        // Search power groups from LARGEST to SMALLEST
        FOR g := 1 TO Num_Unique_Powers DO
            Target_Power_Value := Unique_Powers[g];
            
            // Does this power fit?
            IF Target_Power_Value <= Power_Needed THEN
                // Find available step with this power, lowest cycles
                FOR i := 1 TO Number_Of_Steps DO
                    IF Step_Power_Rating[i] = Target_Power_Value THEN
                        Step_Available := NOT Coil_Internal[i] AND NOT Step_Quarantined[i];
                        
                        IF Step_Available AND Step_Cycle_Count[i] < Min_Cycles THEN
                            Best_Step := i;
                            Min_Cycles := Step_Cycle_Count[i];
                        END_IF;
                    END_IF;
                END_FOR;
                
                // Found a step? Use it
                IF Best_Step > 0 THEN
                    EXIT;
                END_IF;
            END_IF;
        END_FOR;
        
        // If no large step fits, find smallest available step
        IF Best_Step = 0 THEN
            FOR g := Num_Unique_Powers TO 1 BY -1 DO
                Target_Power_Value := Unique_Powers[g];
                
                FOR i := 1 TO Number_Of_Steps DO
                    IF Step_Power_Rating[i] = Target_Power_Value THEN
                        Step_Available := NOT Coil_Internal[i] AND NOT Step_Quarantined[i];
                        
                        IF Step_Available THEN
                            IF Best_Step = 0 OR Step_Cycle_Count[i] < Min_Cycles THEN
                                Best_Step := i;
                                Min_Cycles := Step_Cycle_Count[i];
                            END_IF;
                        END_IF;
                    END_IF;
                END_FOR;
                
                IF Best_Step > 0 THEN
                    EXIT;
                END_IF;
            END_FOR;
        END_IF;
        
        // Turn ON selected step
        IF Best_Step > 0 THEN
            Coil_Internal[Best_Step] := TRUE;
            Step_Cycle_Count[Best_Step] := Step_Cycle_Count[Best_Step] + 1;
        END_IF;
        
        Step_Up_Timer(IN := FALSE);
    END_IF;

// ============================================
// NEED TO REMOVE POWER?
// ============================================
ELSIF Power_Needed < -Deadband_kW THEN
    Step_Down_Timer(IN := TRUE, PT := Step_Down_Delay);
    Step_Up_Timer(IN := FALSE);
    
    IF Step_Down_Timer.Q THEN
        Best_Step := 0;
        Max_Cycles := 0;
        
        // Search power groups from SMALLEST to LARGEST
        FOR g := Num_Unique_Powers TO 1 BY -1 DO
            Target_Power_Value := Unique_Powers[g];
            
            // Does this power fit?
            IF Target_Power_Value <= ABS(Power_Needed) THEN
                // Find ON step with this power, highest cycles
                FOR i := 1 TO Number_Of_Steps DO
                    IF Step_Power_Rating[i] = Target_Power_Value AND Coil_Internal[i] THEN
                        IF Step_Cycle_Count[i] >= Max_Cycles THEN
                            Best_Step := i;
                            Max_Cycles := Step_Cycle_Count[i];
                        END_IF;
                    END_IF;
                END_FOR;
                
                IF Best_Step > 0 THEN
                    EXIT;
                END_IF;
            END_IF;
        END_FOR;
        
        // If no step fits, find smallest ON step
        IF Best_Step = 0 THEN
            FOR g := Num_Unique_Powers TO 1 BY -1 DO
                Target_Power_Value := Unique_Powers[g];
                
                FOR i := 1 TO Number_Of_Steps DO
                    IF Step_Power_Rating[i] = Target_Power_Value AND Coil_Internal[i] THEN
                        Best_Step := i;
                        EXIT;
                    END_IF;
                END_FOR;
                
                IF Best_Step > 0 THEN
                    EXIT;
                END_IF;
            END_FOR;
        END_IF;
        
        // Turn OFF selected step
        IF Best_Step > 0 THEN
            Coil_Internal[Best_Step] := FALSE;
        END_IF;
        
        Step_Down_Timer(IN := FALSE);
    END_IF;

ELSE
    // At target - reset timers
    Step_Up_Timer(IN := FALSE);
    Step_Down_Timer(IN := FALSE);
END_IF;

END_IF; // End of non-maintenance mode

// ============================================
// FEEDBACK MONITORING
// ============================================
Any_Feedback_Fault := FALSE;

IF Enable_Feedback_Monitoring THEN
    FOR i := 1 TO Number_Of_Steps DO
        // Reset timer on rising edge (coil just turned ON)
        IF Coil_Internal[i] AND NOT Coil_Prev[i] THEN
            FB_Timer[i](IN := FALSE);
        END_IF;
        
        // Monitor: Coil ON but no feedback
        FB_Timer[i](
            IN := Coil_Internal[i] AND NOT Step_Feedback[i] AND NOT FB_Fault_Latched[i],
            PT := Feedback_Timeout
        );
        
        // Timeout = fault, quarantine step
        IF FB_Timer[i].Q THEN
            FB_Fault_Latched[i] := TRUE;
            Step_Quarantine_Feedback[i] := TRUE;
            Coil_Internal[i] := FALSE;
        END_IF;
        
        IF FB_Fault_Latched[i] THEN
            Any_Feedback_Fault := TRUE;
        END_IF;
        
        Coil_Prev[i] := Coil_Internal[i];
    END_FOR;
END_IF;

// ============================================
// TOTAL POWER MONITORING
// ============================================
IF Enable_Power_Monitoring AND Active_Step_Count > 0 THEN
    // Calculate expected power from ON steps
    Expected_Power := 0.0;
    FOR i := 1 TO Number_Of_Steps DO
        IF Coil_Internal[i] THEN
            Expected_Power := Expected_Power + Step_Power_Rating[i];
        END_IF;
    END_FOR;
    
    // Calculate difference
    Power_Diff := ABS(Measured_Total_Power - Expected_Power);
    
    // Calculate percentage
    IF Expected_Power > 0.0 THEN
        Power_Mismatch_Percent := (Power_Diff / Expected_Power) * 100.0;
    ELSE
        Power_Mismatch_Percent := 0.0;
    END_IF;
    
    // Check if outside tolerance
    Power_Monitor_Timer(
        IN := Power_Mismatch_Percent > Power_Tolerance_Percent,
        PT := Power_Monitor_Delay
    );
    
    IF Power_Monitor_Timer.Q THEN
        Total_Power_Warning := TRUE;
    ELSIF Power_Mismatch_Percent <= Power_Tolerance_Percent THEN
        Total_Power_Warning := FALSE;
        Power_Monitor_Timer(IN := FALSE);
    END_IF;
ELSE
    Power_Monitor_Timer(IN := FALSE);
    Power_Mismatch_Percent := 0.0;
END_IF;

// ============================================
// COPY TO OUTPUT
// ============================================
FOR i := 1 TO LB_NUMBER_OF_STEPS DO
    Step_Coil_Cmd[i] := Coil_Internal[i];
END_FOR;

// ============================================
// CALCULATE RELEASED POWER (final)
// ============================================
Released_Power_kW := 0.0;
Active_Step_Count := 0;
FOR i := 1 TO Number_Of_Steps DO
    IF Coil_Internal[i] THEN
        Released_Power_kW := Released_Power_kW + Step_Power_Rating[i];
        Active_Step_Count := Active_Step_Count + 1;
    END_IF;
END_FOR;

// ============================================
// STATUS MESSAGE
// ============================================
IF Total_Power_Warning THEN
    Status_Text := 'POWER MISMATCH WARNING';
ELSIF Any_Feedback_Fault THEN
    Status_Text := 'FEEDBACK FAULT';
ELSIF Maintenance_Mode THEN
    Status_Text := 'Maintenance mode';
ELSIF At_Target THEN
    Status_Text := 'At target';
ELSIF Power_Needed > 0.0 THEN
    Status_Text := 'Increasing load';
ELSIF Power_Needed < 0.0 THEN
    Status_Text := 'Decreasing load';
ELSE
    Status_Text := 'Ready';
END_IF;

END_FUNCTION_BLOCK

// ---- POUs/FB_Mode_Manager.TcPOU
FUNCTION_BLOCK FB_Mode_Manager
VAR_INPUT
    Mode_Select             : UINT;
    Master_Enable           : BOOL;
    Emergency_Active        : BOOL;
    System_Ready            : BOOL;
END_VAR
VAR_OUTPUT
    Active_Mode             : UINT;
    Mode_Name               : STRING(30);
    Mode_Ready              : BOOL;
    Enable_Output           : BOOL;
END_VAR
VAR
    Mode_Select_Prev        : UINT;
END_VAR

// Emergency forces OFF mode
IF Emergency_Active THEN
    Active_Mode := LB_MODE_OFF;
    Mode_Name := 'EMERGENCY STOP';
    Mode_Ready := FALSE;
    Enable_Output := FALSE;
    RETURN;
END_IF;

// Master enable check
IF NOT Master_Enable THEN
    Active_Mode := LB_MODE_OFF;
    Mode_Name := 'OFF - Enable Required';
    Mode_Ready := FALSE;
    Enable_Output := FALSE;
    RETURN;
END_IF;

// Mode selection
IF Mode_Select <> Mode_Select_Prev THEN
    Active_Mode := Mode_Select;
END_IF;
Mode_Select_Prev := Mode_Select;

// Mode names and enable logic
CASE Active_Mode OF
    LB_MODE_OFF:
        Mode_Name := 'OFF';
        Mode_Ready := TRUE;
        Enable_Output := FALSE;
    
    LB_MODE_AUTO_LEVELING:
        Mode_Name := 'AUTO LOAD LEVELING';
        Mode_Ready := System_Ready;
        Enable_Output := System_Ready;
    
    LB_MODE_NUMERIC:
        Mode_Name := 'NUMERIC LOAD CONTROL';
        Mode_Ready := System_Ready;
        Enable_Output := System_Ready;
    
    LB_MODE_REVERSE_POWER:
        Mode_Name := 'REVERSE POWER';
        Mode_Ready := System_Ready;
        Enable_Output := System_Ready;
    
    LB_MODE_MANUAL:
        Mode_Name := 'MANUAL SWITCH CONTROL';
        Mode_Ready := System_Ready;
        Enable_Output := System_Ready;
    
    LB_MODE_RECIPE:
        Mode_Name := 'RECIPE MODE';
        Mode_Ready := System_Ready;
        Enable_Output := System_Ready;
    
    LB_MODE_MAINTENANCE:
        Mode_Name := 'MAINTENANCE MODE';
        Mode_Ready := TRUE;
        Enable_Output := TRUE;
    
    ELSE
        Mode_Name := 'UNKNOWN MODE';
        Mode_Ready := FALSE;
        Enable_Output := FALSE;
        Active_Mode := LB_MODE_OFF;
END_CASE;

END_FUNCTION_BLOCK

// ---- POUs/FB_DataLogger.TcPOU
FUNCTION_BLOCK FB_DataLogger
(******************************************************************************
 * FB_DataLogger
 * 
 * Purpose: Data logging for Load Bank system
 *   1. Circular buffer for HMI trends (real-time viewing)
 *   2. USB/SD CSV file logging (long-term storage)
 *
 * Features:
 *   - Configurable sample rate (1s to 60s)
 *   - Configurable buffer size (up to 3600 samples)
 *   - Daily CSV files with auto-rotation
 *   - Enable/disable for buffer and USB separately
 *
 * Author: Load Bank Project
 * Date: January 2026
 ******************************************************************************)

VAR_INPUT
    // Enable controls
    Enable                  : BOOL := TRUE;         // Master enable
    USB_Log_Enable          : BOOL := TRUE;         // Enable USB file logging
    
    // Sample rate (from GVL_Persistent)
    Sample_Time             : TIME := T#10s;        // How often to sample
    Buffer_Size             : UINT := 360;          // Active buffer size (max 3600)
    
    // Data inputs - Power
    Power_Released          : REAL;
    Power_Target            : REAL;
    
    // Data inputs - Temperature (up to 4 TCs)
    Temp_TC1                : REAL;
    Temp_TC2                : REAL;
    Temp_TC3                : REAL;
    Temp_TC4                : REAL;
    Number_Of_TCs           : UINT := 2;            // How many TCs configured
    
    // Data inputs - Voltage (3-phase)
    Voltage_L1L2            : REAL;
    Voltage_L2L3            : REAL;
    Voltage_L3L1            : REAL;
    
    // Data inputs - Current (3-phase)
    Current_I1              : REAL;
    Current_I2              : REAL;
    Current_I3              : REAL;
    
    // USB path configuration
    USB_Path                : STRING(100) := 'C:\DataLog\';  // Path for CSV files
    
    // Commands
    Clear_Buffer            : BOOL;                 // Clear all trend buffers
    
END_VAR

VAR_OUTPUT
    // Status
    Buffer_Index            : UINT;                 // Current write position (0 to Buffer_Size-1)
    Buffer_Full             : BOOL;                 // Buffer has wrapped at least once
    Samples_Logged          : UDINT;                // Total samples since enable
    
    // USB status
    USB_Active              : BOOL;                 // USB logging is active
    USB_File_Open           : BOOL;                 // File currently open
    USB_Error               : BOOL;                 // Error writing to USB
    USB_Error_Code          : UDINT;                // Last error code
    Current_File_Name       : STRING(50);           // Current log file name
    
    // Trend buffer outputs (circular buffers)
    // These are written to GVL arrays for HMI access
    Trend_Write_Index       : UINT;                 // Current write index for HMI
    
END_VAR

VAR
    // Timing
    Sample_Timer            : TON;
    Sample_Trigger          : BOOL;
    
    // Buffer management
    Internal_Index          : UINT := 0;
    Buffer_Wrapped          : BOOL := FALSE;
    
    // USB file handling
    FB_FileOpen             : FB_FileOpen;
    FB_FilePuts             : FB_FilePuts;
    FB_FileClose            : FB_FileClose;
    FB_CreateDir            : FB_CreateDir;
    
    File_Handle             : UINT := 0;
    File_State              : UINT := 0;            // State machine for file ops
    Write_Buffer            : STRING(500);          // Line buffer for CSV
    
    // Date tracking for daily files
    Last_Day                : WORD := 0;
    Last_Month              : WORD := 0;
    System_Time             : TIMESTRUCT;
    FB_GetTime              : NT_GetTime;
    
    // Internal flags
    Init_Done               : BOOL := FALSE;
    Dir_Created             : BOOL := FALSE;
    Need_New_File           : BOOL := FALSE;
    Write_Pending           : BOOL := FALSE;
    Close_Pending           : BOOL := FALSE;
    
    // Helpers
    i                       : UINT;
    sTemp                   : STRING(20);
    
END_VAR

VAR CONSTANT
    MAX_BUFFER              : UINT := 3600;         // Maximum array size
END_VAR

// ============================================================================
// INITIALIZATION
// ============================================================================
IF NOT Init_Done THEN
    Internal_Index := 0;
    Buffer_Wrapped := FALSE;
    Samples_Logged := 0;
    File_State := 0;
    Init_Done := TRUE;
END_IF

// ============================================================================
// CLEAR BUFFER COMMAND
// ============================================================================
IF Clear_Buffer THEN
    Internal_Index := 0;
    Buffer_Wrapped := FALSE;
    Samples_Logged := 0;
    
    // Clear all GVL trend arrays
    FOR i := 1 TO MAX_BUFFER DO
        Trend_Power_Released[i] := 0.0;
        Trend_Power_Target[i] := 0.0;
        Trend_Temp_TC1[i] := 0.0;
        Trend_Temp_TC2[i] := 0.0;
        Trend_Temp_TC3[i] := 0.0;
        Trend_Temp_TC4[i] := 0.0;
        Trend_Voltage_L1L2[i] := 0.0;
        Trend_Voltage_L2L3[i] := 0.0;
        Trend_Voltage_L3L1[i] := 0.0;
        Trend_Current_I1[i] := 0.0;
        Trend_Current_I2[i] := 0.0;
        Trend_Current_I3[i] := 0.0;
    END_FOR
END_IF

// ============================================================================
// SAMPLE TIMER
// ============================================================================
Sample_Timer(
    IN := Enable AND NOT Sample_Timer.Q,
    PT := Sample_Time
);

Sample_Trigger := Sample_Timer.Q;

// Reset timer on trigger
IF Sample_Trigger THEN
    Sample_Timer(IN := FALSE);
END_IF

// ============================================================================
// GET CURRENT TIME (for file naming and timestamps)
// ============================================================================
FB_GetTime(
    NETID := '',
    START := TRUE,
    TMOUT := T#1s
);

IF NOT FB_GetTime.BUSY AND NOT FB_GetTime.ERR THEN
    System_Time := FB_GetTime.TIMESTR;
END_IF

// ============================================================================
// DATA SAMPLING - CIRCULAR BUFFER
// ============================================================================
IF Enable AND Sample_Trigger THEN
    
    // Clamp buffer size
    IF Buffer_Size > MAX_BUFFER THEN
        Buffer_Size := MAX_BUFFER;
    END_IF
    IF Buffer_Size < 1 THEN
        Buffer_Size := 1;
    END_IF
    
    // Calculate array index (1-based for TwinCAT arrays)
    i := Internal_Index + 1;
    
    // Write to GVL trend arrays
    Trend_Power_Released[i] := Power_Released;
    Trend_Power_Target[i] := Power_Target;
    Trend_Temp_TC1[i] := Temp_TC1;
    Trend_Temp_TC2[i] := Temp_TC2;
    Trend_Temp_TC3[i] := Temp_TC3;
    Trend_Temp_TC4[i] := Temp_TC4;
    Trend_Voltage_L1L2[i] := Voltage_L1L2;
    Trend_Voltage_L2L3[i] := Voltage_L2L3;
    Trend_Voltage_L3L1[i] := Voltage_L3L1;
    Trend_Current_I1[i] := Current_I1;
    Trend_Current_I2[i] := Current_I2;
    Trend_Current_I3[i] := Current_I3;
    
    // Increment index with wrap-around
    Internal_Index := Internal_Index + 1;
    IF Internal_Index >= Buffer_Size THEN
        Internal_Index := 0;
        Buffer_Wrapped := TRUE;
    END_IF
    
    // Update outputs
    Buffer_Index := Internal_Index;
    Buffer_Full := Buffer_Wrapped;
    Samples_Logged := Samples_Logged + 1;
    Trend_Write_Index := Internal_Index;
    
    // Trigger USB write
    IF USB_Log_Enable THEN
        Write_Pending := TRUE;
    END_IF
    
END_IF

// ============================================================================
// USB FILE LOGGING - STATE MACHINE
// ============================================================================
IF USB_Log_Enable AND Enable THEN
    
    CASE File_State OF
        
        // --------------------------------------------------------------------
        // State 0: Idle / Check if new file needed
        // --------------------------------------------------------------------
        0:
            USB_Active := TRUE;
            
            // Check if date changed (need new daily file)
            IF (System_Time.wDay <> Last_Day) OR (System_Time.wMonth <> Last_Month) OR NOT USB_File_Open THEN
                Need_New_File := TRUE;
                
                // Close existing file first if open
                IF USB_File_Open THEN
                    File_State := 50;  // Go to close state
                ELSE
                    File_State := 10;  // Go to create directory
                END_IF
            ELSIF Write_Pending THEN
                File_State := 30;  // Go to write state
            END_IF
            
        // --------------------------------------------------------------------
        // State 10: Create directory if needed
        // --------------------------------------------------------------------
        10:
            FB_CreateDir(
                sNetId := '',
                sPathName := USB_Path,
                ePath := PATH_GENERIC,
                bExecute := TRUE,
                tTimeout := T#2s
            );
            File_State := 11;
            
        11:
            FB_CreateDir(bExecute := FALSE);
            IF NOT FB_CreateDir.bBusy THEN
                // Ignore error (directory may already exist)
                Dir_Created := TRUE;
                File_State := 20;  // Go to open file
            END_IF
            
        // --------------------------------------------------------------------
        // State 20: Open/Create daily CSV file
        // --------------------------------------------------------------------
        20:
            // Build filename: YYYY-MM-DD.csv
            Current_File_Name := CONCAT(
                CONCAT(
                    CONCAT(
                        CONCAT(USB_Path, WORD_TO_STRING(System_Time.wYear)),
                        '-'
                    ),
                    RIGHT(CONCAT('0', WORD_TO_STRING(System_Time.wMonth)), 2)
                ),
                CONCAT(
                    CONCAT('-', RIGHT(CONCAT('0', WORD_TO_STRING(System_Time.wDay)), 2)),
                    '.csv'
                )
            );
            
            FB_FileOpen(
                sNetId := '',
                sPathName := Current_File_Name,
                nMode := FOPEN_MODEAPPEND OR FOPEN_MODETEXT,
                ePath := PATH_GENERIC,
                bExecute := TRUE,
                tTimeout := T#2s
            );
            File_State := 21;
            
        21:
            FB_FileOpen(bExecute := FALSE);
            IF NOT FB_FileOpen.bBusy THEN
                IF FB_FileOpen.bError THEN
                    USB_Error := TRUE;
                    USB_Error_Code := FB_FileOpen.nErrId;
                    File_State := 0;
                ELSE
                    File_Handle := FB_FileOpen.hFile;
                    USB_File_Open := TRUE;
                    USB_Error := FALSE;
                    Last_Day := System_Time.wDay;
                    Last_Month := System_Time.wMonth;
                    Need_New_File := FALSE;
                    
                    // Write header if new file (check file position)
                    File_State := 25;
                END_IF
            END_IF
            
        // --------------------------------------------------------------------
        // State 25: Write CSV header (for new files)
        // --------------------------------------------------------------------
        25:
            // CSV Header line
            Write_Buffer := 'Timestamp,Power_Released,Power_Target,Temp_TC1,Temp_TC2,Temp_TC3,Temp_TC4,Voltage_L1L2,Voltage_L2L3,Voltage_L3L1,Current_I1,Current_I2,Current_I3';
            Write_Buffer := CONCAT(Write_Buffer, '$n');
            
            FB_FilePuts(
                sNetId := '',
                hFile := File_Handle,
                sLine := Write_Buffer,
                bExecute := TRUE,
                tTimeout := T#1s
            );
            File_State := 26;
            
        26:
            FB_FilePuts(bExecute := FALSE);
            IF NOT FB_FilePuts.bBusy THEN
                IF FB_FilePuts.bError THEN
                    USB_Error := TRUE;
                    USB_Error_Code := FB_FilePuts.nErrId;
                END_IF
                File_State := 0;  // Back to idle
            END_IF
            
        // --------------------------------------------------------------------
        // State 30: Write data line
        // --------------------------------------------------------------------
        30:
            IF NOT USB_File_Open THEN
                File_State := 10;  // Need to open file first
            ELSE
                // Build CSV line: Timestamp,Data1,Data2,...
                // Timestamp format: YYYY-MM-DD HH:MM:SS
                Write_Buffer := CONCAT(
                    CONCAT(
                        CONCAT(WORD_TO_STRING(System_Time.wYear), '-'),
                        CONCAT(RIGHT(CONCAT('0', WORD_TO_STRING(System_Time.wMonth)), 2), '-')
                    ),
                    CONCAT(
                        RIGHT(CONCAT('0', WORD_TO_STRING(System_Time.wDay)), 2),
                        ' '
                    )
                );
                Write_Buffer := CONCAT(Write_Buffer,
                    CONCAT(
                        CONCAT(RIGHT(CONCAT('0', WORD_TO_STRING(System_Time.wHour)), 2), ':'),
                        CONCAT(
                            CONCAT(RIGHT(CONCAT('0', WORD_TO_STRING(System_Time.wMinute)), 2), ':'),
                            RIGHT(CONCAT('0', WORD_TO_STRING(System_Time.wSecond)), 2)
                        )
                    )
                );
                
                // Add data values
                Write_Buffer := CONCAT(Write_Buffer, ',');
                Write_Buffer := CONCAT(Write_Buffer, REAL_TO_STRING(Power_Released));
                Write_Buffer := CONCAT(Write_Buffer, ',');
                Write_Buffer := CONCAT(Write_Buffer, REAL_TO_STRING(Power_Target));
                Write_Buffer := CONCAT(Write_Buffer, ',');
                Write_Buffer := CONCAT(Write_Buffer, REAL_TO_STRING(Temp_TC1));
                Write_Buffer := CONCAT(Write_Buffer, ',');
                Write_Buffer := CONCAT(Write_Buffer, REAL_TO_STRING(Temp_TC2));
                Write_Buffer := CONCAT(Write_Buffer, ',');
                Write_Buffer := CONCAT(Write_Buffer, REAL_TO_STRING(Temp_TC3));
                Write_Buffer := CONCAT(Write_Buffer, ',');
                Write_Buffer := CONCAT(Write_Buffer, REAL_TO_STRING(Temp_TC4));
                Write_Buffer := CONCAT(Write_Buffer, ',');
                Write_Buffer := CONCAT(Write_Buffer, REAL_TO_STRING(Voltage_L1L2));
                Write_Buffer := CONCAT(Write_Buffer, ',');
                Write_Buffer := CONCAT(Write_Buffer, REAL_TO_STRING(Voltage_L2L3));
                Write_Buffer := CONCAT(Write_Buffer, ',');
                Write_Buffer := CONCAT(Write_Buffer, REAL_TO_STRING(Voltage_L3L1));
                Write_Buffer := CONCAT(Write_Buffer, ',');
                Write_Buffer := CONCAT(Write_Buffer, REAL_TO_STRING(Current_I1));
                Write_Buffer := CONCAT(Write_Buffer, ',');
                Write_Buffer := CONCAT(Write_Buffer, REAL_TO_STRING(Current_I2));
                Write_Buffer := CONCAT(Write_Buffer, ',');
                Write_Buffer := CONCAT(Write_Buffer, REAL_TO_STRING(Current_I3));
                Write_Buffer := CONCAT(Write_Buffer, '$n');
                
                FB_FilePuts(
                    sNetId := '',
                    hFile := File_Handle,
                    sLine := Write_Buffer,
                    bExecute := TRUE,
                    tTimeout := T#1s
                );
                File_State := 31;
            END_IF
            
        31:
            FB_FilePuts(bExecute := FALSE);
            IF NOT FB_FilePuts.bBusy THEN
                IF FB_FilePuts.bError THEN
                    USB_Error := TRUE;
                    USB_Error_Code := FB_FilePuts.nErrId;
                END_IF
                Write_Pending := FALSE;
                File_State := 0;  // Back to idle
            END_IF
            
        // --------------------------------------------------------------------
        // State 50: Close file
        // --------------------------------------------------------------------
        50:
            FB_FileClose(
                sNetId := '',
                hFile := File_Handle,
                bExecute := TRUE,
                tTimeout := T#2s
            );
            File_State := 51;
            
        51:
            FB_FileClose(bExecute := FALSE);
            IF NOT FB_FileClose.bBusy THEN
                USB_File_Open := FALSE;
                File_Handle := 0;
                
                IF Need_New_File THEN
                    File_State := 10;  // Create new file
                ELSE
                    File_State := 0;   // Back to idle
                END_IF
            END_IF
            
    END_CASE
    
ELSE
    // USB logging disabled
    USB_Active := FALSE;
    
    // Close file if open
    IF USB_File_Open THEN
        File_State := 50;
    END_IF
    
END_IF

// ============================================================================
// DISABLE HANDLING
// ============================================================================
IF NOT Enable THEN
    Sample_Timer(IN := FALSE);
    USB_Active := FALSE;
    
    // Close file on disable
    IF USB_File_Open AND File_State = 0 THEN
        File_State := 50;
    END_IF
END_IF

END_FUNCTION_BLOCK

// ---- POUs/FB_Alarm_Manager.TcPOU
FUNCTION_BLOCK FB_Alarm_Manager
// ============================================
// FB_Alarm_Manager
// Professional alarm management for Load Bank
// Features:
//   - 17 defined alarms (critical + warning)
//   - Active alarm list with timestamps
//   - Alarm history (last 50 events)
//   - Individual + Acknowledge All
//   - Clear history command
//   - Works with or without RTC
//   - Priority-based status text
// ============================================

VAR_INPUT
    // ============================================
    // ALARM SOURCE SIGNALS (directly from FBs/IO)
    // ============================================
    
    // Emergency (Critical)
    IN_Emergency_Immediate      : BOOL;     // Alarm 1
    IN_Emergency_Controlled     : BOOL;     // Alarm 2
    
    // Temperature (Critical + Warning)
    IN_Temp_Overtemp            : BOOL;     // Alarm 3 - Critical
    IN_Temp_Warning             : BOOL;     // Alarm 4 - Warning
    IN_TC_Sensor_Fail           : BOOL;     // Alarm 5 - Critical
    IN_Inlet_Overtemp           : BOOL;     // Alarm 6 - Critical
    IN_Inlet_TC_Fail            : BOOL;     // Alarm 7 - Critical
    IN_TC_Contingency           : BOOL;     // Alarm 8 - Warning
    
    // Fan (Critical)
    IN_Fan_Motor_Overload       : BOOL;     // Alarm 9
    IN_Fan_Pressure_Fail        : BOOL;     // Alarm 10
    IN_Fan_Contactor_Fail       : BOOL;     // Alarm 11
    
    // Main Contactor (Critical)
    IN_Main_Contactor_Fail      : BOOL;     // Alarm 12
    
    // Load Controller (Critical + Warning)
    IN_Step_Feedback_Fault      : BOOL;     // Alarm 13 - Critical
    IN_Power_Mismatch           : BOOL;     // Alarm 14 - Warning
    
    // Gradual Dump (Critical)
    IN_Dump_Timeout             : BOOL;     // Alarm 15
    
    // Imbalance (Warning)
    IN_Voltage_Imbalance        : BOOL;     // Alarm 16
    IN_Current_Imbalance        : BOOL;     // Alarm 17
    
    // ============================================
    // REAL-TIME CLOCK (Optional)
    // ============================================
    RTC_Valid                   : BOOL := FALSE;    // TRUE if RTC available
    RTC_Year                    : UINT := 0;
    RTC_Month                   : UINT := 0;
    RTC_Day                     : UINT := 0;
    RTC_Hour                    : UINT := 0;
    RTC_Minute                  : UINT := 0;
    RTC_Second                  : UINT := 0;
    
    // ============================================
    // COMMANDS
    // ============================================
    Acknowledge_Alarm           : ARRAY[1..20] OF BOOL;     // Ack individual alarm
    Acknowledge_All_Cmd         : BOOL;                     // Ack all alarms
    Reset_Cmd                   : BOOL;                     // Reset/clear inactive ack'd alarms
    Clear_History_Cmd           : BOOL;                     // Clear history buffer
    
    Enable                      : BOOL := TRUE;
END_VAR

VAR_OUTPUT
    // ============================================
    // SUMMARY FLAGS
    // ============================================
    General_Alarm               : BOOL;     // Any critical alarm active
    General_Warning             : BOOL;     // Any warning active (no critical)
    System_Normal               : BOOL;     // No alarms or warnings
    Any_Fault_Active            : BOOL;     // Blocks Master Enable
    
    // ============================================
    // COUNTS
    // ============================================
    Critical_Alarm_Count        : UINT;     // Number of critical alarms
    Warning_Count               : UINT;     // Number of warnings
    Total_Active_Count          : UINT;     // Total active alarms
    Unacknowledged_Count        : UINT;     // Needs operator attention
    
    // ============================================
    // HMI STATUS BAR
    // ============================================
    Status_Text                 : STRING(100);  // Main status message
    Detail_Text                 : STRING(100);  // Secondary detail
    
    // ============================================
    // ACTIVE ALARM LIST (for HMI table)
    // ============================================
    Alarm_List                  : ARRAY[1..20] OF DUT_Alarm;
    Alarm_List_Count            : UINT;     // How many in list
    
    // ============================================
    // HISTORY (for HMI history tab)
    // ============================================
    Alarm_History               : ARRAY[1..50] OF DUT_Alarm_History_Record;
    History_Count               : UINT;     // Total records in history
    History_Index               : UINT;     // Current write position
    
    // ============================================
    // LED OUTPUTS
    // ============================================
    LED_Alarm                   : BOOL;     // Red LED
    LED_Warning                 : BOOL;     // Yellow LED
    LED_Normal                  : BOOL;     // Green LED
    
    // ============================================
    // NEWEST ALARM (for popup/notification)
    // ============================================
    New_Alarm_Trigger           : BOOL;     // Pulse when new alarm
    Newest_Alarm_ID             : UINT;     // Which alarm just triggered
    Newest_Alarm_Name           : STRING(30);
END_VAR

VAR
    // ============================================
    // ALARM DEFINITIONS (constant data)
    // ============================================
    Alarm_Name                  : ARRAY[1..17] OF STRING(30) := [
        'IMMEDIATE E-STOP',         // 1
        'CONTROLLED E-STOP',        // 2
        'TEMPERATURE CRITICAL',     // 3
        'TEMPERATURE WARNING',      // 4
        'TC SENSOR FAIL',           // 5
        'INLET TEMP HIGH',          // 6
        'INLET TC FAIL',            // 7
        'TC CONTINGENCY MODE',      // 8
        'FAN MOTOR OVERLOAD',       // 9
        'FAN PRESSURE FAIL',        // 10
        'FAN CONTACTOR FAIL',       // 11
        'MAIN CONTACTOR FAIL',      // 12
        'STEP FEEDBACK FAULT',      // 13
        'POWER MISMATCH',           // 14
        'DUMP TIMEOUT',             // 15
        'VOLTAGE IMBALANCE',        // 16
        'CURRENT IMBALANCE'         // 17
    ];
    
    Alarm_Description           : ARRAY[1..17] OF STRING(50) := [
        'All outputs OFF - Reset required',             // 1
        'Controlled shutdown in progress',              // 2
        'Outlet temperature exceeded maximum',          // 3
        'Outlet temperature approaching limit',         // 4
        'Thermocouple open or shorted',                 // 5
        'Inlet/ambient temperature too high',           // 6
        'Inlet thermocouple failed',                    // 7
        'Running with reduced TC monitoring',           // 8
        'Fan motor thermal overload tripped',           // 9
        'Fan pressure not established',                 // 10
        'Fan contactor feedback timeout',               // 11
        'Main contactor feedback timeout',              // 12
        'Load step feedback mismatch',                  // 13
        'Measured power differs from expected',         // 14
        'Gradual dump did not complete in time',        // 15
        'Phase voltage imbalance detected',             // 16
        'Phase current imbalance detected'              // 17
    ];
    
    Alarm_Severity              : ARRAY[1..17] OF UINT := [
        1,  // 1 - Critical
        1,  // 2 - Critical
        1,  // 3 - Critical
        2,  // 4 - Warning
        1,  // 5 - Critical
        1,  // 6 - Critical
        1,  // 7 - Critical
        2,  // 8 - Warning
        1,  // 9 - Critical
        1,  // 10 - Critical
        1,  // 11 - Critical
        1,  // 12 - Critical
        1,  // 13 - Critical
        2,  // 14 - Warning
        1,  // 15 - Critical
        2,  // 16 - Warning
        2   // 17 - Warning
    ];
    
    // ============================================
    // INTERNAL STATE
    // ============================================
    Alarm_Active                : ARRAY[1..17] OF BOOL;     // Current state
    Alarm_Active_Prev           : ARRAY[1..17] OF BOOL;     // Previous scan
    Alarm_Acknowledged          : ARRAY[1..17] OF BOOL;     // Ack state per alarm
    Alarm_Timestamp             : ARRAY[1..17] OF STRING(20);   // When occurred
    Alarm_Start_Time            : ARRAY[1..17] OF UDINT;    // Runtime when started (for duration)
    
    // Runtime counter (if no RTC)
    Runtime_Timer               : TON;
    Runtime_Seconds             : UDINT;    // Seconds since power-on
    Runtime_Days                : UDINT;
    Runtime_Hours               : UINT;
    Runtime_Minutes             : UINT;
    Runtime_Secs                : UINT;
    
    // Working variables
    i                           : UINT;
    j                           : UINT;
    List_Index                  : UINT;
    Highest_Priority_Alarm      : UINT;
    Temp_Alarm                  : DUT_Alarm;
    Temp_History                : DUT_Alarm_History_Record;
    Current_Timestamp           : STRING(20);
    
    // Edge detection
    Ack_All_Prev                : BOOL;
    Reset_Prev                  : BOOL;
    Clear_History_Prev          : BOOL;
    New_Alarm_Pulse             : BOOL;
    
    // First scan
    First_Scan                  : BOOL := TRUE;
END_VAR

// ============================================
// FIRST SCAN - INITIALIZE
// ============================================
IF First_Scan THEN
    FOR i := 1 TO 17 DO
        Alarm_Active[i] := FALSE;
        Alarm_Active_Prev[i] := FALSE;
        Alarm_Acknowledged[i] := FALSE;
        Alarm_Timestamp[i] := '';
        Alarm_Start_Time[i] := 0;
    END_FOR
    
    FOR i := 1 TO 20 DO
        Alarm_List[i].ID := 0;
        Alarm_List[i].Active := FALSE;
    END_FOR
    
    FOR i := 1 TO 50 DO
        Alarm_History[i].Alarm_ID := 0;
    END_FOR
    
    History_Index := 0;
    History_Count := 0;
    First_Scan := FALSE;
END_IF

// ============================================
// NOT ENABLED
// ============================================
IF NOT Enable THEN
    General_Alarm := FALSE;
    General_Warning := FALSE;
    System_Normal := TRUE;
    LED_Alarm := FALSE;
    LED_Warning := FALSE;
    LED_Normal := TRUE;
    Status_Text := 'Alarm Manager Disabled';
    Detail_Text := '';
    RETURN;
END_IF

// ============================================
// RUNTIME COUNTER (for non-RTC timestamp)
// ============================================
Runtime_Timer(IN := TRUE, PT := T#1s);
IF Runtime_Timer.Q THEN
    Runtime_Timer(IN := FALSE);
    Runtime_Seconds := Runtime_Seconds + 1;
END_IF

// Calculate days, hours, minutes, seconds
Runtime_Days := Runtime_Seconds / 86400;
Runtime_Hours := UDINT_TO_UINT((Runtime_Seconds MOD 86400) / 3600);
Runtime_Minutes := UDINT_TO_UINT((Runtime_Seconds MOD 3600) / 60);
Runtime_Secs := UDINT_TO_UINT(Runtime_Seconds MOD 60);

// ============================================
// GENERATE CURRENT TIMESTAMP
// ============================================
IF RTC_Valid THEN
    // Format: "YYYY-MM-DD HH:MM:SS"
    Current_Timestamp := UINT_TO_STRING(RTC_Year);
    Current_Timestamp := CONCAT(Current_Timestamp, '-');
    IF RTC_Month < 10 THEN
        Current_Timestamp := CONCAT(Current_Timestamp, '0');
    END_IF
    Current_Timestamp := CONCAT(Current_Timestamp, UINT_TO_STRING(RTC_Month));
    Current_Timestamp := CONCAT(Current_Timestamp, '-');
    IF RTC_Day < 10 THEN
        Current_Timestamp := CONCAT(Current_Timestamp, '0');
    END_IF
    Current_Timestamp := CONCAT(Current_Timestamp, UINT_TO_STRING(RTC_Day));
    Current_Timestamp := CONCAT(Current_Timestamp, ' ');
    IF RTC_Hour < 10 THEN
        Current_Timestamp := CONCAT(Current_Timestamp, '0');
    END_IF
    Current_Timestamp := CONCAT(Current_Timestamp, UINT_TO_STRING(RTC_Hour));
    Current_Timestamp := CONCAT(Current_Timestamp, ':');
    IF RTC_Minute < 10 THEN
        Current_Timestamp := CONCAT(Current_Timestamp, '0');
    END_IF
    Current_Timestamp := CONCAT(Current_Timestamp, UINT_TO_STRING(RTC_Minute));
    Current_Timestamp := CONCAT(Current_Timestamp, ':');
    IF RTC_Second < 10 THEN
        Current_Timestamp := CONCAT(Current_Timestamp, '0');
    END_IF
    Current_Timestamp := CONCAT(Current_Timestamp, UINT_TO_STRING(RTC_Second));
ELSE
    // Format: "XXXd HH:MM:SS" (runtime)
    Current_Timestamp := UDINT_TO_STRING(Runtime_Days);
    Current_Timestamp := CONCAT(Current_Timestamp, 'd ');
    IF Runtime_Hours < 10 THEN
        Current_Timestamp := CONCAT(Current_Timestamp, '0');
    END_IF
    Current_Timestamp := CONCAT(Current_Timestamp, UINT_TO_STRING(Runtime_Hours));
    Current_Timestamp := CONCAT(Current_Timestamp, ':');
    IF Runtime_Minutes < 10 THEN
        Current_Timestamp := CONCAT(Current_Timestamp, '0');
    END_IF
    Current_Timestamp := CONCAT(Current_Timestamp, UINT_TO_STRING(Runtime_Minutes));
    Current_Timestamp := CONCAT(Current_Timestamp, ':');
    IF Runtime_Secs < 10 THEN
        Current_Timestamp := CONCAT(Current_Timestamp, '0');
    END_IF
    Current_Timestamp := CONCAT(Current_Timestamp, UINT_TO_STRING(Runtime_Secs));
END_IF

// ============================================
// MAP INPUT SIGNALS TO ALARM ARRAY
// ============================================
Alarm_Active[1] := IN_Emergency_Immediate;
Alarm_Active[2] := IN_Emergency_Controlled;
Alarm_Active[3] := IN_Temp_Overtemp;
Alarm_Active[4] := IN_Temp_Warning;
Alarm_Active[5] := IN_TC_Sensor_Fail;
Alarm_Active[6] := IN_Inlet_Overtemp;
Alarm_Active[7] := IN_Inlet_TC_Fail;
Alarm_Active[8] := IN_TC_Contingency;
Alarm_Active[9] := IN_Fan_Motor_Overload;
Alarm_Active[10] := IN_Fan_Pressure_Fail;
Alarm_Active[11] := IN_Fan_Contactor_Fail;
Alarm_Active[12] := IN_Main_Contactor_Fail;
Alarm_Active[13] := IN_Step_Feedback_Fault;
Alarm_Active[14] := IN_Power_Mismatch;
Alarm_Active[15] := IN_Dump_Timeout;
Alarm_Active[16] := IN_Voltage_Imbalance;
Alarm_Active[17] := IN_Current_Imbalance;

// ============================================
// DETECT NEW ALARMS (rising edge)
// ============================================
New_Alarm_Trigger := FALSE;
FOR i := 1 TO 17 DO
    IF Alarm_Active[i] AND NOT Alarm_Active_Prev[i] THEN
        // NEW ALARM - record timestamp
        Alarm_Timestamp[i] := Current_Timestamp;
        Alarm_Start_Time[i] := Runtime_Seconds;
        Alarm_Acknowledged[i] := FALSE;
        
        // Trigger new alarm notification
        New_Alarm_Trigger := TRUE;
        Newest_Alarm_ID := i;
        Newest_Alarm_Name := Alarm_Name[i];
    END_IF
END_FOR

// ============================================
// DETECT CLEARED ALARMS (falling edge) - ADD TO HISTORY
// ============================================
FOR i := 1 TO 17 DO
    IF NOT Alarm_Active[i] AND Alarm_Active_Prev[i] THEN
        // ALARM CLEARED - add to history
        History_Index := History_Index + 1;
        IF History_Index > 50 THEN
            History_Index := 1;     // Circular buffer wrap
        END_IF
        IF History_Count < 50 THEN
            History_Count := History_Count + 1;
        END_IF
        
        Alarm_History[History_Index].Alarm_ID := i;
        Alarm_History[History_Index].Alarm_Name := Alarm_Name[i];
        Alarm_History[History_Index].Severity := Alarm_Severity[i];
        Alarm_History[History_Index].Time_Occurred := Alarm_Timestamp[i];
        Alarm_History[History_Index].Time_Cleared := Current_Timestamp;
        Alarm_History[History_Index].Duration_Sec := Runtime_Seconds - Alarm_Start_Time[i];
        Alarm_History[History_Index].Was_Acknowledged := Alarm_Acknowledged[i];
        
        // Clear timestamp for this alarm
        Alarm_Timestamp[i] := '';
        Alarm_Acknowledged[i] := FALSE;
    END_IF
END_FOR

// Update previous state
FOR i := 1 TO 17 DO
    Alarm_Active_Prev[i] := Alarm_Active[i];
END_FOR

// ============================================
// ACKNOWLEDGE INDIVIDUAL ALARMS
// ============================================
FOR i := 1 TO 17 DO
    IF i <= 20 THEN
        IF Acknowledge_Alarm[i] AND Alarm_Active[i] THEN
            Alarm_Acknowledged[i] := TRUE;
        END_IF
    END_IF
END_FOR

// ============================================
// ACKNOWLEDGE ALL (rising edge)
// ============================================
IF Acknowledge_All_Cmd AND NOT Ack_All_Prev THEN
    FOR i := 1 TO 17 DO
        IF Alarm_Active[i] THEN
            Alarm_Acknowledged[i] := TRUE;
        END_IF
    END_FOR
END_IF
Ack_All_Prev := Acknowledge_All_Cmd;

// ============================================
// CLEAR HISTORY (rising edge)
// ============================================
IF Clear_History_Cmd AND NOT Clear_History_Prev THEN
    FOR i := 1 TO 50 DO
        Alarm_History[i].Alarm_ID := 0;
        Alarm_History[i].Alarm_Name := '';
        Alarm_History[i].Severity := 0;
        Alarm_History[i].Time_Occurred := '';
        Alarm_History[i].Time_Cleared := '';
        Alarm_History[i].Duration_Sec := 0;
        Alarm_History[i].Was_Acknowledged := FALSE;
    END_FOR
    History_Index := 0;
    History_Count := 0;
END_IF
Clear_History_Prev := Clear_History_Cmd;

// ============================================
// COUNT ALARMS
// ============================================
Critical_Alarm_Count := 0;
Warning_Count := 0;
Unacknowledged_Count := 0;

FOR i := 1 TO 17 DO
    IF Alarm_Active[i] THEN
        IF Alarm_Severity[i] = 1 THEN
            Critical_Alarm_Count := Critical_Alarm_Count + 1;
        ELSE
            Warning_Count := Warning_Count + 1;
        END_IF
        
        IF NOT Alarm_Acknowledged[i] THEN
            Unacknowledged_Count := Unacknowledged_Count + 1;
        END_IF
    END_IF
END_FOR

Total_Active_Count := Critical_Alarm_Count + Warning_Count;

// ============================================
// BUILD ACTIVE ALARM LIST (for HMI)
// ============================================
List_Index := 0;

// First add critical alarms (higher priority)
FOR i := 1 TO 17 DO
    IF Alarm_Active[i] AND Alarm_Severity[i] = 1 THEN
        List_Index := List_Index + 1;
        IF List_Index <= 20 THEN
            Alarm_List[List_Index].ID := i;
            Alarm_List[List_Index].Name := Alarm_Name[i];
            Alarm_List[List_Index].Description := Alarm_Description[i];
            Alarm_List[List_Index].Severity := Alarm_Severity[i];
            Alarm_List[List_Index].Active := TRUE;
            Alarm_List[List_Index].Acknowledged := Alarm_Acknowledged[i];
            Alarm_List[List_Index].Timestamp_Occurred := Alarm_Timestamp[i];
        END_IF
    END_IF
END_FOR

// Then add warnings
FOR i := 1 TO 17 DO
    IF Alarm_Active[i] AND Alarm_Severity[i] = 2 THEN
        List_Index := List_Index + 1;
        IF List_Index <= 20 THEN
            Alarm_List[List_Index].ID := i;
            Alarm_List[List_Index].Name := Alarm_Name[i];
            Alarm_List[List_Index].Description := Alarm_Description[i];
            Alarm_List[List_Index].Severity := Alarm_Severity[i];
            Alarm_List[List_Index].Active := TRUE;
            Alarm_List[List_Index].Acknowledged := Alarm_Acknowledged[i];
            Alarm_List[List_Index].Timestamp_Occurred := Alarm_Timestamp[i];
        END_IF
    END_IF
END_FOR

Alarm_List_Count := List_Index;

// Clear unused slots
FOR i := List_Index + 1 TO 20 DO
    Alarm_List[i].ID := 0;
    Alarm_List[i].Name := '';
    Alarm_List[i].Active := FALSE;
END_FOR

// ============================================
// SET SUMMARY FLAGS
// ============================================
General_Alarm := Critical_Alarm_Count > 0;
General_Warning := (Warning_Count > 0) AND NOT General_Alarm;
System_Normal := (Total_Active_Count = 0);
Any_Fault_Active := General_Alarm;

// ============================================
// LED OUTPUTS
// ============================================
LED_Alarm := General_Alarm;
LED_Warning := General_Warning;
LED_Normal := System_Normal;

// ============================================
// STATUS TEXT (priority-based)
// ============================================
IF Total_Active_Count = 0 THEN
    Status_Text := 'SYSTEM NORMAL';
    Detail_Text := 'No active alarms';
ELSE
    // Find highest priority (lowest ID among critical)
    Highest_Priority_Alarm := 0;
    FOR i := 1 TO 17 DO
        IF Alarm_Active[i] AND Alarm_Severity[i] = 1 THEN
            IF Highest_Priority_Alarm = 0 THEN
                Highest_Priority_Alarm := i;
            END_IF
        END_IF
    END_FOR
    
    // If no critical, find first warning
    IF Highest_Priority_Alarm = 0 THEN
        FOR i := 1 TO 17 DO
            IF Alarm_Active[i] AND Alarm_Severity[i] = 2 THEN
                IF Highest_Priority_Alarm = 0 THEN
                    Highest_Priority_Alarm := i;
                END_IF
            END_IF
        END_FOR
    END_IF
    
    // Set status text
    IF Highest_Priority_Alarm > 0 THEN
        Status_Text := Alarm_Name[Highest_Priority_Alarm];
        Detail_Text := Alarm_Description[Highest_Priority_Alarm];
    END_IF
    
    // Append count if multiple alarms
    IF Total_Active_Count > 1 THEN
        Status_Text := CONCAT(Status_Text, ' (+');
        Status_Text := CONCAT(Status_Text, UINT_TO_STRING(Total_Active_Count - 1));
        Status_Text := CONCAT(Status_Text, ' more)');
    END_IF
END_IF

END_FUNCTION_BLOCK

// ---- POUs/FB_Auto_Mode.TcPOU
FUNCTION_BLOCK FB_Auto_Mode
VAR_INPUT
    Mode_Active             : BOOL;
    External_Power_kW       : REAL;             // From external power meter
    Min_Load_kW             : REAL;             // Minimum load to maintain on generator
    Available_Power_kW      : REAL;             // Max available from Load_Controller
    Deadband_kW             : REAL := 5.0;      // Default 5 kW deadband
    System_Ready            : BOOL;
END_VAR

VAR_OUTPUT
    Target_Power_kW         : REAL;             // Target for Load_Controller
    Power_Error             : REAL;             // For HMI display
    Status_Text             : STRING(100);      // Status for HMI
END_VAR

VAR
    Internal_Target         : REAL;
END_VAR

// ============================================
// NOT ACTIVE - IDLE
// ============================================
IF NOT Mode_Active THEN
    Target_Power_kW := 0.0;
    Power_Error := 0.0;
    Status_Text := 'Mode not active';
    RETURN;
END_IF;

// ============================================
// SYSTEM NOT READY
// ============================================
IF NOT System_Ready THEN
    Target_Power_kW := 0.0;
    Power_Error := 0.0;
    Status_Text := 'System not ready';
    RETURN;
END_IF;

// ============================================
// AUTO LEVELING ALGORITHM
// ============================================
// Power_Error = How far external power is from target (Min_Load_kW)
// Positive error = too much power flowing out, need to remove load
// Negative error = reverse power or under target, need to add load
Power_Error := External_Power_kW - Min_Load_kW;

// Calculate new target
Internal_Target := Target_Power_kW - Power_Error;

// Clamp to valid range
IF Internal_Target < 0.0 THEN
    Internal_Target := 0.0;
ELSIF Internal_Target > Available_Power_kW THEN
    Internal_Target := Available_Power_kW;
END_IF;

Target_Power_kW := Internal_Target;

// ============================================
// STATUS TEXT
// ============================================
IF ABS(Power_Error) <= Deadband_kW THEN
    Status_Text := 'At target';
ELSIF Power_Error < -Deadband_kW THEN
    // Need to add load
    IF Target_Power_kW >= Available_Power_kW THEN
        Status_Text := 'LB FULL - Cannot add more';
    ELSE
        Status_Text := 'Adding load';
    END_IF;
ELSE
    // Need to remove load
    IF Target_Power_kW <= 0.0 THEN
        Status_Text := 'LB Empty - Cannot remove more';
    ELSE
        Status_Text := 'Removing load';
    END_IF;
END_IF;

END_FUNCTION_BLOCK

// ---- POUs/FB_Numeric_Mode.TcPOU
FUNCTION_BLOCK FB_Numeric_Mode
VAR_INPUT
    Mode_Active             : BOOL;             // TRUE when this mode is selected
    Target_Power_Setpoint   : REAL;             // User entered kW value from HMI keypad
    Rated_Power_kW          : REAL;             // Load bank rated capacity (limit)
    System_Ready            : BOOL;             // System ready to operate
END_VAR

VAR_OUTPUT
    Target_Power_kW         : REAL;             // Output to Load_Controller
    Status_Text             : STRING(100);      // Status for HMI
END_VAR

VAR
    Clamped_Target          : REAL;
END_VAR

// ============================================
// NOT ACTIVE - RESET OUTPUT
// ============================================
IF NOT Mode_Active THEN
    Target_Power_kW := 0.0;
    Status_Text := 'Mode not active';
    RETURN;
END_IF;

// ============================================
// SYSTEM NOT READY
// ============================================
IF NOT System_Ready THEN
    Target_Power_kW := 0.0;
    Status_Text := 'System not ready';
    RETURN;
END_IF;

// ============================================
// VALIDATE AND CLAMP TO RATED CAPACITY
// ============================================
Clamped_Target := Target_Power_Setpoint;

// No negative values
IF Clamped_Target < 0.0 THEN
    Clamped_Target := 0.0;
END_IF;

// Limit to rated capacity
IF Clamped_Target > Rated_Power_kW THEN
    Clamped_Target := Rated_Power_kW;
    Status_Text := 'Limited to rated capacity';
ELSIF Clamped_Target = 0.0 THEN
    Status_Text := 'Idle - Enter target power';
ELSE
    Status_Text := 'Running';
END_IF;

Target_Power_kW := Clamped_Target;

END_FUNCTION_BLOCK

// ---- POUs/FB_Reverse_Mode.TcPOU
FUNCTION_BLOCK FB_Reverse_Mode

VAR_INPUT
    Mode_Active             : BOOL;             // TRUE when this mode is selected
    Generator_Power_kW      : REAL;             // Power from external meter (generator output)
    Follow_Percentage       : REAL := 100.0;    // % of generator power to absorb (0-100)
    Max_Power_kW            : REAL;             // Available power limit
    System_Ready            : BOOL;             // System ready to operate
END_VAR

VAR_OUTPUT
    Target_Power_kW         : REAL;             // Output to Load_Controller
    Status_Text             : STRING(100);      // Status for HMI
END_VAR

VAR
    Calculated_Target       : REAL;
    Clamped_Percentage      : REAL;
END_VAR

// ============================================
// NOT ACTIVE - RESET OUTPUT
// ============================================
IF NOT Mode_Active THEN
    Target_Power_kW := 0.0;
    Status_Text := 'Mode not active';
    RETURN;
END_IF;


// ============================================
// SYSTEM NOT READY
// ============================================
IF NOT System_Ready THEN
    Target_Power_kW := 0.0;
    Status_Text := 'System not ready';
    RETURN;
END_IF;


// ============================================
// VALIDATE FOLLOW PERCENTAGE
// ============================================
Clamped_Percentage := Follow_Percentage;

IF Clamped_Percentage < 0.0 THEN
    Clamped_Percentage := 0.0;
ELSIF Clamped_Percentage > 100.0 THEN
    Clamped_Percentage := 100.0;
END_IF;


// ============================================
// CALCULATE TARGET POWER
// ============================================
Calculated_Target := Generator_Power_kW * (Clamped_Percentage / 100.0);


// ============================================
// CLAMP TO AVAILABLE POWER
// ============================================
IF Calculated_Target < 0.0 THEN
    Calculated_Target := 0.0;
END_IF;

IF Calculated_Target > Max_Power_kW THEN
    Calculated_Target := Max_Power_kW;
    Status_Text := 'Limited to available power';
ELSIF Generator_Power_kW <= 0.0 THEN
    Status_Text := 'Waiting for generator power';
ELSIF Clamped_Percentage = 0.0 THEN
    Status_Text := 'Follow at 0% - No load';
ELSE
    Status_Text := 'Following generator';
END_IF;


// ============================================
// OUTPUT
// ============================================
Target_Power_kW := Calculated_Target;

END_FUNCTION_BLOCK

// ---- POUs/FB_Manual_Mode.TcPOU
FUNCTION_BLOCK FB_Manual_Mode
VAR_INPUT
    Number_Of_Switches      : USINT;
    Switch_Status           : ARRAY[1..8] OF BOOL;
    Switch_Power            : ARRAY[1..8] OF REAL;
END_VAR
VAR_OUTPUT
    Target_Power_kW         : REAL;
END_VAR
VAR
    i                       : USINT;
END_VAR

Target_Power_kW := 0.0;

FOR i := 1 TO Number_Of_Switches DO
    IF Switch_Status[i] THEN
        Target_Power_kW := Target_Power_kW + Switch_Power[i];
    END_IF;
END_FOR;

END_FUNCTION_BLOCK

// ---- POUs/FB_Recipe_Controller.TcPOU
FUNCTION_BLOCK FB_Recipe_Controller
VAR_INPUT
    Recipe_Enable           : BOOL;
    Recipe_Start            : BOOL;
    Recipe_Pause            : BOOL;
    Recipe_Abort            : BOOL;
    
    Recipe_Steps            : ARRAY[1..20] OF DUT_Recipe_Step;
    Number_Of_Steps         : UINT := 5;
    
    Current_Power_kW        : REAL;
END_VAR
VAR_OUTPUT
    Recipe_Running          : BOOL;
    Recipe_Paused           : BOOL;
    Recipe_Complete         : BOOL;
    Recipe_Aborted          : BOOL;
    
    Current_Step_Number     : UINT;
    Current_Step_Name       : STRING(40);
    Target_Power_kW         : REAL;
    
    Step_Elapsed_Time       : TIME;
    Step_Remaining_Time     : TIME;
    
    Total_Recipe_Time       : TIME;
    Total_Elapsed_Time      : TIME;
    Total_Remaining_Time    : TIME;
    
    Recipe_Progress_Percent : UINT;
    
    Status_Message          : STRING(100);
END_VAR
VAR
    State                   : UINT;
    Step_Timer              : TON;
    Elapsed_Total           : TIME;
    
    Recipe_Start_Prev       : BOOL;
    Recipe_Pause_Prev       : BOOL;
    Recipe_Abort_Prev       : BOOL;
    
    i                       : UINT;
END_VAR



IF NOT Recipe_Enable THEN
    State := 0;
    Recipe_Running := FALSE;
    Recipe_Paused := FALSE;
    Target_Power_kW := 0.0;
    RETURN;
END_IF;

// Calculate total recipe time
Total_Recipe_Time := T#0s;
FOR i := 1 TO Number_Of_Steps DO
    IF Recipe_Steps[i].Enabled THEN
        Total_Recipe_Time := Total_Recipe_Time + Recipe_Steps[i].Duration;
    END_IF;
END_FOR;

CASE State OF
    0: // IDLE
        Recipe_Running := FALSE;
        Recipe_Paused := FALSE;
        Recipe_Complete := FALSE;
        Recipe_Aborted := FALSE;
        
        Current_Step_Number := 0;
        Current_Step_Name := '';
        Target_Power_kW := 0.0;
        
        Step_Elapsed_Time := T#0s;
        Total_Elapsed_Time := T#0s;
        Elapsed_Total := T#0s;
        
        Status_Message := 'Recipe idle - press START';
        
        Step_Timer(IN := FALSE);
        
        IF Recipe_Start AND NOT Recipe_Start_Prev THEN
            Current_Step_Number := 1;
            State := 10;
        END_IF;
    
    10: // RUNNING
        Recipe_Running := TRUE;
        Recipe_Paused := FALSE;
        Recipe_Complete := FALSE;
        Recipe_Aborted := FALSE;
        
        IF Current_Step_Number > Number_Of_Steps OR Current_Step_Number = 0 THEN
            State := 90;
            RETURN;
        END_IF;
        
        IF NOT Recipe_Steps[Current_Step_Number].Enabled THEN
            Current_Step_Number := Current_Step_Number + 1;
            RETURN;
        END_IF;
        
        Current_Step_Name := Recipe_Steps[Current_Step_Number].Step_Name;
        Target_Power_kW := Recipe_Steps[Current_Step_Number].Target_Power_kW;
        
        Step_Timer(IN := TRUE, PT := Recipe_Steps[Current_Step_Number].Duration);
        
        Step_Elapsed_Time := Step_Timer.ET;
        Step_Remaining_Time := Recipe_Steps[Current_Step_Number].Duration - Step_Timer.ET;
        
        Elapsed_Total := Elapsed_Total + T#100ms;
        Total_Elapsed_Time := Elapsed_Total;
        Total_Remaining_Time := Total_Recipe_Time - Elapsed_Total;
        
        IF Total_Recipe_Time > T#0s THEN
            Recipe_Progress_Percent := DINT_TO_UINT((TIME_TO_DINT(Elapsed_Total) * 100) / TIME_TO_DINT(Total_Recipe_Time));
        ELSE
            Recipe_Progress_Percent := 0;
        END_IF;
        
        Status_Message := CONCAT('Running step ', UINT_TO_STRING(Current_Step_Number));
        Status_Message := CONCAT(Status_Message, ': ');
        Status_Message := CONCAT(Status_Message, Current_Step_Name);
        
        IF Recipe_Pause AND NOT Recipe_Pause_Prev THEN
            State := 20;
        END_IF;
        
        IF Recipe_Abort AND NOT Recipe_Abort_Prev THEN
            State := 99;
        END_IF;
        
        IF Step_Timer.Q THEN
            Current_Step_Number := Current_Step_Number + 1;
            Step_Timer(IN := FALSE);
            
            IF Current_Step_Number > Number_Of_Steps THEN
                State := 90;
            END_IF;
        END_IF;
    
    20: // PAUSED
        Recipe_Running := FALSE;
        Recipe_Paused := TRUE;
        
        Step_Timer(IN := FALSE);
        
        Status_Message := 'Recipe PAUSED';
        
        IF Recipe_Start AND NOT Recipe_Start_Prev THEN
            State := 10;
        END_IF;
        
        IF Recipe_Abort AND NOT Recipe_Abort_Prev THEN
            State := 99;
        END_IF;
    
    90: // COMPLETE
        Recipe_Running := FALSE;
        Recipe_Paused := FALSE;
        Recipe_Complete := TRUE;
        Recipe_Aborted := FALSE;
        
        Target_Power_kW := 0.0;
        
        Status_Message := 'Recipe COMPLETE';
        
        Step_Timer(IN := FALSE);
        
        IF Recipe_Start AND NOT Recipe_Start_Prev THEN
            State := 0;
        END_IF;
    
    99: // ABORTED
        Recipe_Running := FALSE;
        Recipe_Paused := FALSE;
        Recipe_Complete := FALSE;
        Recipe_Aborted := TRUE;
        
        Target_Power_kW := 0.0;
        
        Status_Message := 'Recipe ABORTED by operator';
        
        Step_Timer(IN := FALSE);
        
        IF Recipe_Start AND NOT Recipe_Start_Prev THEN
            State := 0;
        END_IF;
        
END_CASE;

Recipe_Start_Prev := Recipe_Start;
Recipe_Pause_Prev := Recipe_Pause;
Recipe_Abort_Prev := Recipe_Abort;

END_FUNCTION_BLOCK

// ---- POUs/FB_Maintenance_Mode.TcPOU
FUNCTION_BLOCK FB_Maintenance_Mode
VAR_INPUT
    Mode_Active             : BOOL;
    
    Number_of_Steps         : UINT := 10;
    
    Test_Step_Number        : UINT;
    Test_Fan_Command        : BOOL;
    Test_Step_Command       : BOOL;
    
    Step_Feedback           : ARRAY[1..100] OF BOOL;
    Fan_Running             : BOOL;
    
    Master_Enable           : BOOL;
    Emergency_Active        : BOOL;
END_VAR
VAR_OUTPUT
    Mode_Ready              : BOOL;
    Test_Active             : BOOL;
    
    Step_Output             : ARRAY[1..100] OF BOOL;
    Fan_Start               : BOOL;
    
    Status_Message          : STRING(100);
    Fault_Message           : STRING(100);
END_VAR
VAR
    i                       : UINT;
    Test_Step_Prev          : BOOL;
    Test_Fan_Prev           : BOOL;
END_VAR



IF NOT Mode_Active THEN
    Test_Active := FALSE;
    Mode_Ready := FALSE;
    
    FOR i := 1 TO 100 DO
        Step_Output[i] := FALSE;
    END_FOR;
    
    Fan_Start := FALSE;
    Status_Message := 'Maintenance mode not active';
    Fault_Message := '';
    RETURN;
END_IF;

IF Emergency_Active THEN
    Test_Active := FALSE;
    Mode_Ready := FALSE;
    
    FOR i := 1 TO 100 DO
        Step_Output[i] := FALSE;
    END_FOR;
    
    Fan_Start := FALSE;
    Status_Message := 'EMERGENCY ACTIVE';
    Fault_Message := 'Emergency stop activated';
    RETURN;
END_IF;

IF NOT Master_Enable THEN
    Mode_Ready := FALSE;
    Status_Message := 'Master enable required';
    Fault_Message := '';
    RETURN;
END_IF;

Mode_Ready := TRUE;

// Fan test
IF Test_Fan_Command AND NOT Test_Fan_Prev THEN
    Fan_Start := NOT Fan_Start;
    
    IF Fan_Start THEN
        Status_Message := 'Fan test ACTIVE';
    ELSE
        Status_Message := 'Fan test STOPPED';
    END_IF;
END_IF;

Test_Fan_Prev := Test_Fan_Command;

// Step test
IF Test_Step_Command AND NOT Test_Step_Prev THEN
    IF Test_Step_Number > 0 AND Test_Step_Number <= Number_of_Steps THEN
        Step_Output[Test_Step_Number] := NOT Step_Output[Test_Step_Number];
        
        IF Step_Output[Test_Step_Number] THEN
            Test_Active := TRUE;
            Status_Message := CONCAT('Testing step ', UINT_TO_STRING(Test_Step_Number));
            Status_Message := CONCAT(Status_Message, ' - ON');
        ELSE
            Test_Active := FALSE;
            Status_Message := CONCAT('Testing step ', UINT_TO_STRING(Test_Step_Number));
            Status_Message := CONCAT(Status_Message, ' - OFF');
        END_IF;
    ELSE
        Fault_Message := 'Invalid step number';
    END_IF;
END_IF;

Test_Step_Prev := Test_Step_Command;

// Check feedback
IF Test_Active THEN
    IF Test_Step_Number > 0 AND Test_Step_Number <= Number_of_Steps THEN
        IF Step_Output[Test_Step_Number] AND NOT Step_Feedback[Test_Step_Number] THEN
            Fault_Message := CONCAT('Step ', UINT_TO_STRING(Test_Step_Number));
            Fault_Message := CONCAT(Fault_Message, ' feedback fault');
        ELSIF NOT Step_Output[Test_Step_Number] AND Step_Feedback[Test_Step_Number] THEN
            Fault_Message := CONCAT('Step ', UINT_TO_STRING(Test_Step_Number));
            Fault_Message := CONCAT(Fault_Message, ' contactor stuck');
        ELSE
            Fault_Message := '';
        END_IF;
    END_IF;
END_IF;

END_FUNCTION_BLOCK

// ---- POUs/FB_Recipe_Storage_Manager.TcPOU
FUNCTION_BLOCK FB_Recipe_Storage_Manager
VAR_INPUT
    // Commands from HMI
    Save_Recipe             : BOOL;
    Load_Recipe             : BOOL;
    Delete_Recipe           : BOOL;
    
    // Which slot to operate on
    Selected_Slot           : UINT;             // 1-4
    
    // Current recipe data to save
    Current_Recipe_Name     : STRING(40);
    Current_Steps           : ARRAY[1..20] OF DUT_Recipe_Step;
    Current_Number_Of_Steps : UINT;
END_VAR

VAR_OUTPUT
    // Loaded recipe data
    Loaded_Recipe_Name      : STRING(40);
    Loaded_Steps            : ARRAY[1..20] OF DUT_Recipe_Step;
    Loaded_Number_Of_Steps  : UINT;
    
    // Status
    Operation_Complete      : BOOL;
    Operation_Status        : STRING(50);
    
    // Recipe slot info for HMI display
    Slot_1_Name             : STRING(40);
    Slot_1_Valid            : BOOL;
    Slot_2_Name             : STRING(40);
    Slot_2_Valid            : BOOL;
    Slot_3_Name             : STRING(40);
    Slot_3_Valid            : BOOL;
    Slot_4_Name             : STRING(40);
    Slot_4_Valid            : BOOL;
END_VAR

VAR
    Save_Prev               : BOOL;
    Load_Prev               : BOOL;
    Delete_Prev             : BOOL;
    
    i                       : UINT;
    TotalTime               : TIME;
    MaxPower                : REAL;
END_VAR

// Update slot info for HMI display
Slot_1_Name := GVL_Recipe_Storage.Saved_Recipes[1].Recipe_Name;
Slot_1_Valid := GVL_Recipe_Storage.Saved_Recipes[1].Is_Valid;
Slot_2_Name := GVL_Recipe_Storage.Saved_Recipes[2].Recipe_Name;
Slot_2_Valid := GVL_Recipe_Storage.Saved_Recipes[2].Is_Valid;
Slot_3_Name := GVL_Recipe_Storage.Saved_Recipes[3].Recipe_Name;
Slot_3_Valid := GVL_Recipe_Storage.Saved_Recipes[3].Is_Valid;
Slot_4_Name := GVL_Recipe_Storage.Saved_Recipes[4].Recipe_Name;
Slot_4_Valid := GVL_Recipe_Storage.Saved_Recipes[4].Is_Valid;

// Reset operation complete flag
Operation_Complete := FALSE;

// Validate slot selection
IF Selected_Slot < 1 OR Selected_Slot > 4 THEN
    Selected_Slot := 1;
END_IF;


// ==========================================
// SAVE RECIPE
// ==========================================
IF Save_Recipe AND NOT Save_Prev THEN
    
    // Validate we have data to save
    IF Current_Number_Of_Steps > 0 AND Current_Recipe_Name <> '' THEN
        
        // Save recipe name and step count
        GVL_Recipe_Storage.Saved_Recipes[Selected_Slot].Recipe_Name := Current_Recipe_Name;
        GVL_Recipe_Storage.Saved_Recipes[Selected_Slot].Number_Of_Steps := Current_Number_Of_Steps;
        
        // Calculate total duration and peak power
        TotalTime := T#0s;
        MaxPower := 0.0;
        
        FOR i := 1 TO Current_Number_Of_Steps DO
            // Copy step data
            GVL_Recipe_Storage.Saved_Recipes[Selected_Slot].Steps[i] := Current_Steps[i];
            
            // Accumulate time
            IF Current_Steps[i].Enabled THEN
                TotalTime := TotalTime + Current_Steps[i].Duration;
                IF Current_Steps[i].Target_Power_kW > MaxPower THEN
                    MaxPower := Current_Steps[i].Target_Power_kW;
                END_IF;
            END_IF;
        END_FOR;
        
        // Clear remaining steps
        FOR i := Current_Number_Of_Steps + 1 TO 20 DO
            GVL_Recipe_Storage.Saved_Recipes[Selected_Slot].Steps[i].Step_Name := '';
            GVL_Recipe_Storage.Saved_Recipes[Selected_Slot].Steps[i].Target_Power_kW := 0.0;
            GVL_Recipe_Storage.Saved_Recipes[Selected_Slot].Steps[i].Duration := T#0s;
            GVL_Recipe_Storage.Saved_Recipes[Selected_Slot].Steps[i].Enabled := FALSE;
        END_FOR;
        
        // Save calculated values
        GVL_Recipe_Storage.Saved_Recipes[Selected_Slot].Total_Duration := TotalTime;
        GVL_Recipe_Storage.Saved_Recipes[Selected_Slot].Peak_Power_kW := MaxPower;
        GVL_Recipe_Storage.Saved_Recipes[Selected_Slot].Is_Valid := TRUE;
        
        Operation_Status := 'Recipe saved successfully';
        Operation_Complete := TRUE;
        
    ELSE
        Operation_Status := 'Error: No recipe data to save';
        Operation_Complete := TRUE;
    END_IF;
    
END_IF;
Save_Prev := Save_Recipe;


// ==========================================
// LOAD RECIPE
// ==========================================
IF Load_Recipe AND NOT Load_Prev THEN
    
    // Check if slot has valid data
    IF GVL_Recipe_Storage.Saved_Recipes[Selected_Slot].Is_Valid THEN
        
        // Load recipe data
        Loaded_Recipe_Name := GVL_Recipe_Storage.Saved_Recipes[Selected_Slot].Recipe_Name;
        Loaded_Number_Of_Steps := GVL_Recipe_Storage.Saved_Recipes[Selected_Slot].Number_Of_Steps;
        
        // Copy steps
        FOR i := 1 TO 20 DO
            Loaded_Steps[i] := GVL_Recipe_Storage.Saved_Recipes[Selected_Slot].Steps[i];
        END_FOR;
        
        Operation_Status := 'Recipe loaded successfully';
        Operation_Complete := TRUE;
        
    ELSE
        Operation_Status := 'Error: No recipe in selected slot';
        Operation_Complete := TRUE;
    END_IF;
    
END_IF;
Load_Prev := Load_Recipe;


// ==========================================
// DELETE RECIPE
// ==========================================
IF Delete_Recipe AND NOT Delete_Prev THEN
    
    // Clear the selected slot
    GVL_Recipe_Storage.Saved_Recipes[Selected_Slot].Recipe_Name := '';
    GVL_Recipe_Storage.Saved_Recipes[Selected_Slot].Number_Of_Steps := 0;
    GVL_Recipe_Storage.Saved_Recipes[Selected_Slot].Total_Duration := T#0s;
    GVL_Recipe_Storage.Saved_Recipes[Selected_Slot].Peak_Power_kW := 0.0;
    GVL_Recipe_Storage.Saved_Recipes[Selected_Slot].Is_Valid := FALSE;
    
    // Clear all steps
    FOR i := 1 TO 20 DO
        GVL_Recipe_Storage.Saved_Recipes[Selected_Slot].Steps[i].Step_Name := '';
        GVL_Recipe_Storage.Saved_Recipes[Selected_Slot].Steps[i].Target_Power_kW := 0.0;
        GVL_Recipe_Storage.Saved_Recipes[Selected_Slot].Steps[i].Duration := T#0s;
        GVL_Recipe_Storage.Saved_Recipes[Selected_Slot].Steps[i].Enabled := FALSE;
    END_FOR;
    
    Operation_Status := 'Recipe deleted';
    Operation_Complete := TRUE;
    
END_IF;
Delete_Prev := Delete_Recipe;

END_FUNCTION_BLOCK

// ---- POUs/PRG_Maint_Mode.TcPOU
PROGRAM PRG_Maint_Mode
// ============================================
// MAINTENANCE MODE PROGRAM
// Called from PRG_Main
// ============================================

VAR
    // Manual test edge detection
    Toggle_Step_Prev        : BOOL;
    Toggle_Fan_Prev         : BOOL;
    Reset_Test_Prev         : BOOL;
    Self_Test_Start_Prev    : BOOL;
    Self_Test_Stop_Prev     : BOOL;
    
    // Self test state machine
    Self_Test_State         : INT := 0;
    Feedback_Wait_Timer_ms  : INT := 0;
    Delay_Timer_ms          : INT := 0;
    Second_Counter_ms       : INT := 0;
    
    // Cycle time in ms (adjust to your task cycle)
    Cycle_Time_ms           : INT := 10;
END_VAR


// ============================================
// PROGRAM BODY
// ============================================

// Only run when in maintenance mode
IF LB_System_Status.Active_Mode = LB_MODE_MAINTENANCE THEN

    // ========================================
    // MANUAL FAN TOGGLE (rising edge)
    // ========================================
    IF Maint_Mode_Toggle_Fan AND NOT Toggle_Fan_Prev THEN
        IO_Fan_Contactor_Coil := NOT IO_Fan_Contactor_Coil;
    END_IF;
    Toggle_Fan_Prev := Maint_Mode_Toggle_Fan;
    
    // ========================================
    // MANUAL STEP TOGGLE (rising edge)
    // ========================================
    IF Maint_Mode_Toggle_Step AND NOT Toggle_Step_Prev THEN
        // Interlock: Fan must be running
        IF IO_Fan_Contactor_FB AND IO_Fan_Pressure_OK THEN
            IO_Load_Contactor_Coil[Maint_Mode_Selected_Step] := 
                NOT IO_Load_Contactor_Coil[Maint_Mode_Selected_Step];
        END_IF;
    END_IF;
    Toggle_Step_Prev := Maint_Mode_Toggle_Step;
    
    // ========================================
    // RESET TEST (rising edge)
    // ========================================
    IF Maint_Mode_Reset_Test AND NOT Reset_Test_Prev THEN
        IO_Load_Contactor_Coil[Maint_Mode_Selected_Step] := FALSE;
        Maint_Mode_Feedback_Match := TRUE;
        Maint_Mode_Response_Time_ms := 0;
        Maint_Mode_Power_Within_Tolerance := TRUE;
    END_IF;
    Reset_Test_Prev := Maint_Mode_Reset_Test;
    
    // ========================================
    // FEEDBACK MATCH CHECK (continuous)
    // ========================================
    IF IO_Load_Contactor_Coil[Maint_Mode_Selected_Step] THEN
        Maint_Mode_Feedback_Match := 
            IO_Load_Contactor_Coil[Maint_Mode_Selected_Step] = 
            IO_Load_Contactor_FB[Maint_Mode_Selected_Step];
        
        // Power tolerance check
        IF LB_HMI_Steps[Maint_Mode_Selected_Step].Rated_Power_kW > 0 THEN
            Maint_Mode_Power_Within_Tolerance := 
                ABS(LB_HMI_Steps[Maint_Mode_Selected_Step].Power_Error_Percent) 
                <= Maint_Mode_Power_Tolerance_Percent;
        END_IF;
    END_IF;
    
    // ========================================
    // SELF TEST STATE MACHINE
    // ========================================
    
    // Start command (rising edge)
    IF Maint_Mode_Self_Test_Start AND NOT Self_Test_Start_Prev THEN
        IF NOT Maint_Mode_Self_Test_Running THEN
            // Check interlocks
            IF IO_Fan_Contactor_FB AND IO_Fan_Pressure_OK AND NOT IO_Fan_Motor_Overload_OK THEN
                Maint_Mode_Self_Test_Running := TRUE;
                Maint_Mode_Self_Test_Current_Step := 1;
                Maint_Mode_Self_Test_Pass_Count := 0;
                Maint_Mode_Self_Test_Fail_Count := 0;
                Maint_Mode_Self_Test_Complete := FALSE;
                Maint_Mode_Timeout_Error_Count := 0;
                Self_Test_State := 10;
            END_IF;
        END_IF;
    END_IF;
    Self_Test_Start_Prev := Maint_Mode_Self_Test_Start;
    
    // Stop command (rising edge)
    IF Maint_Mode_Self_Test_Stop AND NOT Self_Test_Stop_Prev THEN
        IF Maint_Mode_Self_Test_Running THEN
            IO_Load_Contactor_Coil[Maint_Mode_Self_Test_Current_Step] := FALSE;
            Maint_Mode_Self_Test_Running := FALSE;
            Self_Test_State := 0;
        END_IF;
    END_IF;
    Self_Test_Stop_Prev := Maint_Mode_Self_Test_Stop;
    
    // State machine
    CASE Self_Test_State OF
        
        0: // IDLE
            ; // Do nothing, wait for start
            
        10: // START NEXT STEP
            IF Maint_Mode_Self_Test_Current_Step <= LB_HMI_Total_Steps THEN
                // Skip quarantined steps
                IF LB_HMI_Steps[Maint_Mode_Self_Test_Current_Step].Status_Quarantined THEN
                    Maint_Mode_Self_Test_Current_Step := Maint_Mode_Self_Test_Current_Step + 1;
                ELSE
                    // Start testing this step
                    IO_Load_Contactor_Coil[Maint_Mode_Self_Test_Current_Step] := TRUE;
                    Maint_Mode_Self_Test_Timer_Sec := Maint_Mode_Test_Duration_Sec;
                    Feedback_Wait_Timer_ms := 0;
                    Second_Counter_ms := 0;
                    Self_Test_State := 20;
                END_IF;
            ELSE
                // All steps tested
                Self_Test_State := 100;
            END_IF;
            
        20: // WAIT FOR FEEDBACK
            Feedback_Wait_Timer_ms := Feedback_Wait_Timer_ms + Cycle_Time_ms;
            
            IF IO_Load_Contactor_FB[Maint_Mode_Self_Test_Current_Step] THEN
                // Feedback received
                Maint_Mode_Response_Time_ms := Feedback_Wait_Timer_ms;
                Maint_Mode_Feedback_Match := TRUE;
                Self_Test_State := 30;
            ELSIF Feedback_Wait_Timer_ms > Maint_Mode_Feedback_Timeout_ms THEN
                // Timeout - FAIL
                Maint_Mode_Timeout_Error_Count := Maint_Mode_Timeout_Error_Count + 1;
                Maint_Mode_Feedback_Match := FALSE;
                Self_Test_State := 90;
            END_IF;
            
        30: // MONITOR POWER FOR DURATION
            // Second countdown
            Second_Counter_ms := Second_Counter_ms + Cycle_Time_ms;
            IF Second_Counter_ms >= 1000 THEN
                Second_Counter_ms := 0;
                Maint_Mode_Self_Test_Timer_Sec := Maint_Mode_Self_Test_Timer_Sec - 1;
            END_IF;
            
            // Check power tolerance continuously
            IF LB_HMI_Steps[Maint_Mode_Self_Test_Current_Step].Rated_Power_kW > 0 THEN
                Maint_Mode_Power_Within_Tolerance := 
                    ABS(LB_HMI_Steps[Maint_Mode_Self_Test_Current_Step].Power_Error_Percent) 
                    <= Maint_Mode_Power_Tolerance_Percent;
            END_IF;
            
            // Check feedback still matches
            Maint_Mode_Feedback_Match := 
                IO_Load_Contactor_FB[Maint_Mode_Self_Test_Current_Step];
            
            // Test duration complete?
            IF Maint_Mode_Self_Test_Timer_Sec <= 0 THEN
                IF Maint_Mode_Power_Within_Tolerance AND Maint_Mode_Feedback_Match THEN
                    Self_Test_State := 80; // PASS
                ELSE
                    Self_Test_State := 90; // FAIL
                END_IF;
            END_IF;
            
        80: // STEP PASSED
            LB_HMI_Steps[Maint_Mode_Self_Test_Current_Step].Status_Quarantined := FALSE;
            Maint_Mode_Self_Test_Pass_Count := Maint_Mode_Self_Test_Pass_Count + 1;
            IO_Load_Contactor_Coil[Maint_Mode_Self_Test_Current_Step] := FALSE;
            Delay_Timer_ms := 0;
            Self_Test_State := 85;
            
        85: // DELAY BEFORE NEXT STEP
            Delay_Timer_ms := Delay_Timer_ms + Cycle_Time_ms;
            IF Delay_Timer_ms >= 1000 THEN
                Maint_Mode_Self_Test_Current_Step := Maint_Mode_Self_Test_Current_Step + 1;
                Self_Test_State := 10;
            END_IF;
            
        90: // STEP FAILED - QUARANTINE
            LB_HMI_Steps[Maint_Mode_Self_Test_Current_Step].Status_Quarantined := TRUE;
            Maint_Mode_Self_Test_Fail_Count := Maint_Mode_Self_Test_Fail_Count + 1;
            LB_HMI_Quarantined_Count := LB_HMI_Quarantined_Count + 1;
            IO_Load_Contactor_Coil[Maint_Mode_Self_Test_Current_Step] := FALSE;
            Delay_Timer_ms := 0;
            Self_Test_State := 85;
            
        100: // ALL STEPS COMPLETE
            Maint_Mode_Self_Test_Running := FALSE;
            Maint_Mode_Self_Test_Complete := TRUE;
            Self_Test_State := 0;
            
    END_CASE;

ELSE
    // ========================================
    // NOT IN MAINTENANCE MODE - Safety reset
    // ========================================
    IF Maint_Mode_Self_Test_Running THEN
        IO_Load_Contactor_Coil[Maint_Mode_Self_Test_Current_Step] := FALSE;
        Maint_Mode_Self_Test_Running := FALSE;
        Self_Test_State := 0;
    END_IF;
    
END_IF;

END_PROGRAM

// ---- GlobalTextList.TcGTLO
TEXTLIST GlobalTextList
  549 = '%t'
  250 = 'EMERGENCY'
  375 = 'FAN'
  911 = 'Fan'
  533 = 'Fan:'
  881 = 'LOAD BANK CONTROL - 480VAC'
  906 = 'Running'
  935 = 'RUNNING'
  693 = 'TEMP'
  861 = 'Temp'
  534 = 'Temp:'
END_TEXTLIST
